TYPE ST_KeyValuePair : 
STRUCT
	sKey: WSTRING(127);
	sValue: STRING(255);
END_STRUCT
END_TYPE

(* stored: DUT ST_KeyValuePair: Id cb73c14d-52a3-4a92-997d-70026272edfb *)
